// TwinCAT 3 PLC project CycleManagerTest
// ProgramVersion: 3.1.4026.19
// libraries:
//   CNM_AbstractObject, * (ekvip automation GmbH)
//   CNM_CommandInterfaces, * (ekvip automation GmbH)
//   CNM_CycleManager, * (ekvip automation GmbH)
//   CNM_CycleManagerInterfaces, * (ekvip automation GmbH)
//   CNM_CycleManagerInterfacesTests, * (ekvip automation GmbH)
//   CNM_ReturnTypes, * (ekvip automation GmbH)
//   Tc2_Standard, * (Beckhoff Automation GmbH)
//   Tc2_System, * (Beckhoff Automation GmbH)
//   TcUnit, * (www.tcunit.org)
// project tree:
//   / PlcTask.TcTTO
//   Tasks/ MAIN.TcPOU
// real-time tasks:
//   TASK PlcTask: cycle T#10ms, priority 20, ADS port 350

CONFIGURATION CycleManagerTest
    RESOURCE PLC ON TwinCAT3
        TASK PlcTask(INTERVAL := T#10ms, PRIORITY := 20);
        PROGRAM MAIN WITH PlcTask : MAIN;
    END_RESOURCE
END_CONFIGURATION

// ---- Tasks/MAIN.TcPOU
PROGRAM MAIN
VAR
	cycleManager :CNM_CycleManager.SimpleCycleManager;
	interfaceTests :CNM_CycleManagerInterfacesTests.InterfaceTests(cycleManager);
END_VAR

TcUnit.RUN();

END_PROGRAM
